TYPE BreakStopConfig :
STRUCT
	MaxTimeLeavingStop :	TIME;				
	DebounceTimePuckPresentOn :	TIME;				
	DebounceTimePuckPresentOff : TIME;			
	DebounceTimeBufferFullOn :	TIME;			
	DebounceTimeBufferFullOff :	TIME;			
	TimeSpacingMinimum	:	TIME;				
	EnableBufferArrivalFault :	BOOL;
	BufferArrivalFaultTime	: TIME;				
END_STRUCT
END_TYPE

(* stored: Version 1.1.0.1, ProductVersion 3.1.4024.6
   DUT BreakStopConfig: Id {31aa5792-7b49-4306-9996-d472e518c42e} *)
